Staubli VAL3: setEventNoWait.pgx

public program setEventNoWait(num handle_, num event_, bool& result_[])
begin
  // set event without wait
  nCommand[handle_]=coSE
  call sendCommand(handle_,"se"+toString("0.0",event_),result_)
end
